PROGRAM P_Inputs
VAR
	fbJoystick 				: FB_JoystickInputScaling;
	fbPositionSensor 		: FB_PositionInputScaling;
	fbPressureSupplySensor 	: FB_PressureInputScaling;
	fbPressureReturnSensor 	: FB_PressureInputScaling;
	fbPressurePistonSide 	: FB_PressureInputScaling;
	fbPressureLhvSide 		: FB_PressureInputScaling;
	fbPressureRodSide 		: FB_PressureInputScaling;
END_VAR

fbJoystick(
	bEnable := G_Inputs.bManualModeSelector,
	nRawInput := G_Inputs.stJoyY.nValue,
	fOutput => G_Sensors.fJoystickY
);

fbPositionSensor(
	nRawInput := G_Inputs.stCylPos.nValue,
	fOutput => G_Sensors.fPistonPosition
);

fbPressureSupplySensor(
	nRawInput := G_Inputs.stPressureSupply.nValue,
	fOutput => G_Sensors.fPressureSupply
);

fbPressureReturnSensor(
	nRawInput := G_Inputs.stPressureReturn.nValue,
	fOutput => G_Sensors.fPressureReturn
);

fbPressurePistonSide(
	nRawInput := G_Inputs.stPressurePistonSide.nValue,
	fOutput => G_Sensors.fPressurePistonSide
);

fbPressureLhvSide(
	nRawInput := G_Inputs.stPressureLhvSide.nValue,
	fOutput => G_Sensors.fPressureLhvSide
);

fbPressureRodSide(
	nRawInput := G_Inputs.stPressureRodSide.nValue,
	fOutput => G_Sensors.fPressureRodSide
);

END_PROGRAM

(* stored: Version 1.1.0.1, ProductVersion 3.1.4024.10
   POU P_Inputs: Id {8b676dbd-393f-42d6-8803-330b6e90ab14}, SpecialFunc None *)
